{attribute 'GeneratedUsingTerminal: EL5101-0000-1019'}
{attribute addProperty BoxType "EL5101-0000-1019"}
{attribute addProperty Id "EtcSlaveTerminalBaseENC_Status_compactAT %I*ENC_Status_compact_D1AA753920ENC_Control_compactAT %Q*ENC_Control_compact_6FDDC6696WcStateAT %I*WcState_9091E0EB2InfoDataAT %I*InfoData_32EB74EA10"}
{attribute addProperty CRC "122766061"}
{attribute addProperty Size "38"}
TYPE EL5101_075142ED EXTENDS EtcSlaveTerminalBase :
STRUCT
	{attribute addProperty Name "ENC_Status_compact"}
	ENC_Status_compact : ENC_Status_compact_D1AA7539;
	{attribute addProperty Name "ENC_Control_compact"}
	ENC_Control_compact : ENC_Control_compact_6FDDC669;
	{attribute addProperty Name "WcState"}
	WcState : WcState_9091E0EB;
	{attribute addProperty Name "InfoData"}
	InfoData : InfoData_32EB74EA;
END_STRUCT
END_TYPE

(* stored: Version 1.2.0.0, ProductVersion 3.1.4024.9
   DUT EL5101_075142ED: Id {2060762e-91a9-4f9d-84df-10fff978dd0b} *)
